FUNCTION Camera_ClearErrors : BOOL
VAR_IN_OUT
	Camera : Cognex_Camera;
END_VAR

IF Camera.CameraState := Camera_State.Error THEN
	Camera.Inspection.Clear_Error := TRUE;
	Camera.CameraState := Camera_State.Clear_Error;
END_IF

END_FUNCTION

(* stored: Version 1.1.0.1, ProductVersion 3.1.4024.10
   POU Camera_ClearErrors: Id {6eb76ee5-3bfd-48d4-b377-858ecb0f5bbc}, SpecialFunc None *)
